// TIA Portal V19 export
TYPE "ValveMachine_PB"
// stored: Access Published
   STRUCT
      Rest : Bool;
      Work : Bool;
      StartStop : Bool;
   END_STRUCT;
END_TYPE
